PROGRAM TESTPRG
VAR
    piper_test : FB_Piper_Test;
    piper_module_test : FB_Piper_Module_Test;
END_VAR

// Copyright (c) 2024 Loupe (https://loupe.team), provided under the MIT License.

TcUnit.RUN();

END_PROGRAM

(* stored: Version 1.1.0.1
   POU TESTPRG: Id {64cf3e97-3804-4926-8187-b690cb96d9b0}, SpecialFunc None *)
